(* PLC project sfc, plcc plcc tests 1 *)
(* stored: creationDateTime 2026-09-27T00:00:00 *)

PROGRAM Sequence
  VAR
    go : BOOL;
  END_VAR

INITIAL_STEP Init:
END_STEP
TRANSITION FROM Init TO ?
  := go;
END_TRANSITION
END_PROGRAM
